DATA_BLOCK "dbArchiveSlotShipping"
{ S7_Optimized_Access := 'TRUE' }
VERSION : 0.8
NON_RETAIN
"fbArchiveSlotShipping"

BEGIN

END_DATA_BLOCK

